# B&R Automation Studio project Robtek17G10
Automation Studio 4.3.3.196

## Configuration Config1

### Task classes (Cpu.sw)
```
Cyclic#7:
  Test <- Test.prg
Binaries: udbdef, TCData, ashwac, arconfig, asfw, ashwd, iomap, User, Role, sysconf
Libraries: runtime, astime, asieccon
```

### Hardware
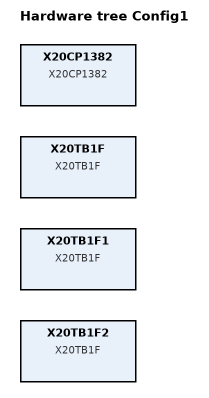
```
X20CP1382 : X20CP1382 v1.3.2.0  [X1 -> X1.SL; X2 -> X2.SL; X3 -> X3.SL]
  Module X1 (Type=X1, Virtual=true, Version=1.3.2.0)
    Connection (Connector=SS1, TargetModule=X20TB1F, TargetConnector=SS)
    Connection (Connector=SL, TargetModule=X20CP1382, TargetConnector=X1)
  Module X2 (Type=X2, Virtual=true, Version=1.3.2.0)
    Connection (Connector=SS1, TargetModule=X20TB1F1, TargetConnector=SS)
    Connection (Connector=SL, TargetModule=X20CP1382, TargetConnector=X2)
  Module X3 (Type=X3, Virtual=true, Version=1.3.2.0)
    Connection (Connector=SS1, TargetModule=X20TB1F2, TargetConnector=SS)
    Connection (Connector=SL, TargetModule=X20CP1382, TargetConnector=X3)
  Connector IF2:
    ActivateDevice = 1
  ConfigurationID = LOS_PETOS
  ConfigVersion = 1.0.1
  UserPartitionSize = 1
  Simulation = 1
  ClearNVMemoryAfterCFChange = 1
  RebootReset = 32
X20TB1F : X20TB1F v1.0.0.0
X20TB1F1 : X20TB1F v1.0.0.0
X20TB1F2 : X20TB1F v1.0.0.0
```

### IoMap.iom - X20CP1382/IoMap.iom
```iecst
VAR_CONFIG
	::x_dir AT %QX."X3".DigitalOutput01;
	::x_en AT %QX."X3".DigitalOutput02;
	::x_step AT %QX."X3".DigitalOutput10;
	::y_step AT %QX."X3".DigitalOutput11;
	::z_step AT %QX."X3".DigitalOutput12;
	::y_dir AT %QX."X3".DigitalOutput03;
	::y_en AT %QX."X3".DigitalOutput04;
	::z_dir AT %QX."X3".DigitalOutput05;
	::z_en AT %QX."X3".DigitalOutput06;
END_VAR
```

## Logical view

### Global.var - Global variables
```iecst
VAR
	x_en : BOOL;
	x_dir : BOOL;
	x_step : BOOL;
	y_en : BOOL;
	y_dir : BOOL;
	y_step : BOOL;
	z_en : BOOL;
	z_dir : BOOL;
	z_step : BOOL;
	stepCount : USINT;
END_VAR
```

### Program Logical/Test (IEC)

#### Main.st - Init, cyclic, exit code
```iecst
PROGRAM _INIT
	//Starter programmet ud med at sætte det hele til at være stille.
	x_dir := FALSE;
	x_en := TRUE;
	x_step := FALSE;

	y_dir := FALSE;
	y_en := TRUE;
	y_step := FALSE;

	z_dir := FALSE;
	z_en := TRUE;
	z_step := FALSE;
	stepCount := 101;
END_PROGRAM

PROGRAM _CYCLIC
	WHILE stepCount > 100 DO
		IF x_step = FALSE THEN
			x_step := TRUE;
		ELSE
			x_step := FALSE;
		END_IF
	END_WHILE

	stepCount := stepCount + 1;
END_PROGRAM

PROGRAM _EXIT
	(* Insert code here *)

END_PROGRAM
```

#### Variables.var - Local variables
```iecst
VAR
	go : BOOL;
END_VAR
```

#### LocalFunctions.fun
```iecst
FUNCTION stepTimes : BOOL
	VAR_INPUT
		x : USINT;
	END_VAR
	VAR_IN_OUT
		u : BOOL;
	END_VAR
	VAR
		b : USINT;
	END_VAR
END_FUNCTION
```

#### Functions.st
```iecst
FUNCTION stepTimes
	FOR b := 1 TO x BY 1 DO
		u := FALSE;
	END_FOR

END_FUNCTION
```

Listed in the project but not available here: Logical/Global.typ, Logical/Libraries, Logical/Test/Types.typ
